(* IEC 61131-3 sources: learning-path/06_oop_in_st/exercises/0_basic_valve_class/test, 1 file *)

(* ---- test.st ---- *)
USING AxUnit;

NAMESPACE MyTest

    {TestFixture}
    CLASS MyTestFixture

        VAR PROTECTED
        END_VAR

        {Test}
        METHOD PUBLIC MyTestMethod
            VAR_TEMP
                result : BOOL;
            END_VAR

            Assert.Equal(actual := FALSE, expected := FALSE);

        END_METHOD
    END_CLASS

END_NAMESPACE
